SYSTEM fbe_testing
  (* Version 1.0, 2024-03-18, cabral *)
  APPLICATION fbe_testingApp
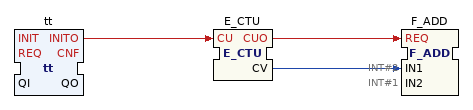
    FBS
      F_ADD : F_ADD(IN1 := INT#2, IN2 := INT#1);
      E_CTU : E_CTU;
    END_FBS
    SUBAPPS
      tt : tt;
    END_SUBAPPS
    EVENT_CONNECTIONS
      E_CTU.CUO TO F_ADD.REQ;
      tt.INITO TO E_CTU.CU;
    END_CONNECTIONS
    DATA_CONNECTIONS
      E_CTU.CV TO F_ADD.IN1;
    END_CONNECTIONS
  END_APPLICATION
  APPLICATION test
  END_APPLICATION
  DEVICE FORTE_PC : FORTE_PC(MGR_ID := "localhost:61499")
    {SET_ATTRIBUTE(Profile, HOLOBLOC)} (* device profile *)
    RESOURCE EMB_RES : EMB_RES
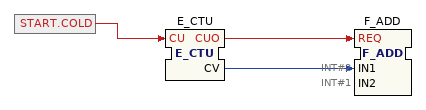
      FBS
        F_ADD : F_ADD(IN1 := INT#2, IN2 := INT#1);
        E_CTU : E_CTU;
      END_FBS
      EVENT_CONNECTIONS
        E_CTU.CUO TO F_ADD.REQ;
        START.COLD TO E_CTU.CU;
      END_CONNECTIONS
      DATA_CONNECTIONS
        E_CTU.CV TO F_ADD.IN1;
      END_CONNECTIONS
    END_RESOURCE
  END_DEVICE
  DEVICE PFC200 : PFC200(MGR_ID := "localhost:61499")
    {SET_ATTRIBUTE(Profile, HOLOBLOC)} (* device profile *)
  END_DEVICE
  MAPPINGS
    fbe_testingApp.F_ADD ON FORTE_PC.EMB_RES.F_ADD;
    fbe_testingApp.E_CTU ON FORTE_PC.EMB_RES.E_CTU;
  END_MAPPINGS
END_SYSTEM
